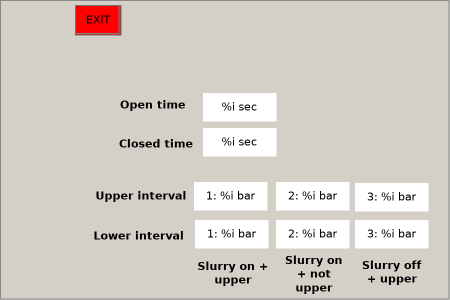
VISUALIZATION LevelControlParamMenu  // 450x300
    Button (75,5 46x30), "EXIT"
        toggle ReactorTemperatureControl.bPIDcontrolParameterMenu
    Label (105,83 100x44), "Open time"
    Label (91,174 100x44), "Upper interval"
    Label (89,214 100x44), "Lower interval"
    Textfield (193,181 75x30), "1: %i bar", text variable: ReactorLevelAndPressureControl.PressureUpperInterVal_1
        OnMouseDown: write the text variable via VisuDialogs.Numpad, min -100, max 100
    Textfield (275,181 75x30), "2: %i bar", text variable: ReactorLevelAndPressureControl.PressureUpperInterVal_2
        OnMouseDown: write the text variable via VisuDialogs.Numpad, min -100, max 100
    Textfield (194,219 75x30), "1: %i bar", text variable: ReactorLevelAndPressureControl.PressureLowerInterval_1
        OnMouseDown: write the text variable via VisuDialogs.Numpad, min -100, max 100
    Textfield (275,219 75x30), "2: %i bar", text variable: ReactorLevelAndPressureControl.PressureLowerInterval_2
        OnMouseDown: write the text variable via VisuDialogs.Numpad, min -100, max 100
    Label (106,122 100x44), "Closed time"
    Textfield (202,92 75x30), "%i sec", text variable: ReactorLevelAndPressureControl.fillingValveOpenInterval
        OnMouseDown: write the text variable via VisuDialogs.Numpad, min 0, max 100
    Textfield (202,127 75x30), "%i sec", text variable: ReactorLevelAndPressureControl.fillingValveCloseInterval
        OnMouseDown: write the text variable via VisuDialogs.Numpad, min 0, max 200
    Textfield (354,182 75x30), "3: %i bar", text variable: ReactorLevelAndPressureControl.PressureUpperInterVal_3
        OnMouseDown: write the text variable via VisuDialogs.Numpad, min -100, max 100
    Textfield (354,219 75x30), "3: %i bar", text variable: ReactorLevelAndPressureControl.PressureLowerInterval_3
        OnMouseDown: write the text variable via VisuDialogs.Numpad, min -100, max 100
    Label (194,251 78x44), "Slurry on + upper"
    Label (356,250 72x44), "Slurry off + upper"
    Label (278,252 72x44), "Slurry on + not upper"
END_VISUALIZATION

(* stored: Version 1.1.0.1, ProductVersion 3.1.4024.9
   Visu LevelControlParamMenu: Id {48d140c7-a1a4-4768-8b33-e23021dc5276} *)
